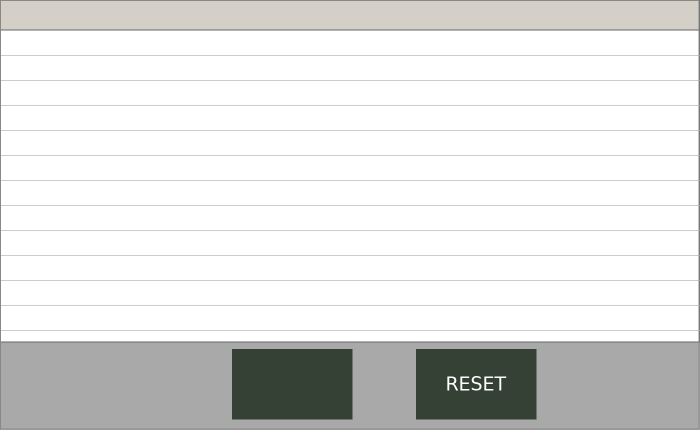
VISUALIZATION E1  // 700x430
    Table (0,0 700x342), data array: GVL_EHS.arrEventVisu
        p3854506369: GVL_EHS.arrEventVisu[INDEX].dwID
        p1892666644: GVL_EHS.arrEventVisu[INDEX].dwParam
        p1218418051: GVL_EHS.arrEventVisu[INDEX].wsMessage
        p746581629: GVL_EHS.arrEventVisu[INDEX].dwColor
        p511219082: Class
        p505689113: Czas ustąpienia
        p3312258591: GVL_EHS.arrEventVisu[INDEX].dwClass
        p2340480326: GVL_EHS.arrEventVisu[INDEX].dtDateEnd
        p1755163831: Opis zdarzenia
        p2237128397: Czas stop
        p2170511999: GVL_EHS.arrEventVisu[INDEX].dtDateBegin
        p4092479075: Czas start
    Rectangle (416,349 120x70), "RESET", colour toggle: GVL_HMI.bResetAlarm
        OnMouseDown: execute { GVL_HMI.bResetAlarm:=TRUE; }
        OnMouseUp: execute { GVL_HMI.bResetAlarm:=FALSE; }
    Rectangle (232,349 120x70), colour toggle: P_EventsVisu.bFilterActiveOnly, text list: 'PrzyciskAlarmy', text index: P_EventsVisu.bFilterActiveOnly
        toggle P_EventsVisu.bFilterActiveOnly
END_VISUALIZATION

(* stored: Version 1.1.0.1, ProductVersion 3.1.4024.15
   Visu E1: Id {dd65c9d5-9011-42b3-afd2-09eb8ec1edb4} *)
